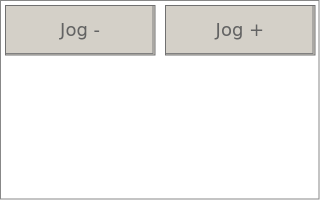
VISUALIZATION SingleAxisJogStandardFlast  // 320x200
VAR_IN_OUT
	btnJogPositive	: BOOL;
	btnJogNegative	: BOOL;
END_VAR
    Button (5,5 150x50), "Jog -"
        tap btnJogNegative
    Button (165,5 150x50), "Jog +"
        tap btnJogPositive
END_VISUALIZATION

(* stored: Version 1.1.0.1, ProductVersion 3.1.4024.9
   Visu SingleAxisJogStandardFlast: Id {fe90b26f-bc31-4a97-9e90-3cec24250cc2} *)
